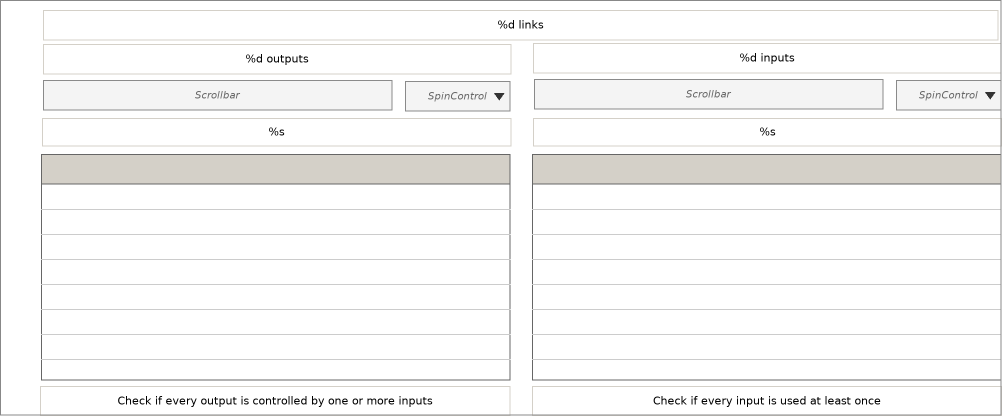
VISUALIZATION LinkInfo  // 1002x416
    Table (41,154 469x226), data array: MAIN.fbHome.stHmi.aLinkedInputs
        p3854506369: MAIN.fbHome.stHmi.aLinkedInputs[INDEX]
        p2232123230: Linked inputs
    Textfield (42,118 469x28), "%s", text variable: MAIN.fbHome.stHmi.sOutput
    SpinControl (405,81 105x30), variable: MAIN.fbHome.stHmi.nOutputIndex
        p651134158: MAIN.fbHome.fbDOGroupAll.nSize-1
    Scrollbar (43,80 349x30)
        p2245068023: MAIN.fbHome.fbDOGroupAll.nSize-1
        p1057716461: MAIN.fbHome.stHmi.nOutputIndex
    Textfield (533,118 469x28), "%s", text variable: MAIN.fbHome.stHmi.sInput
    Scrollbar (534,79 349x30)
        p2245068023: MAIN.fbHome.fbDIGroupAll.nSize-1
        p1057716461: MAIN.fbHome.stHmi.nInputIndex
    SpinControl (896,80 105x30), variable: MAIN.fbHome.stHmi.nInputIndex
        p651134158: MAIN.fbHome.fbDIGroupAll.nSize-1
    Table (532,154 469x226), data array: MAIN.fbHome.stHmi.aLinkedOutputs
        p3854506369: MAIN.fbHome.stHmi.aLinkedOutputs[INDEX]
        p2232123230: Linked outputs
    Textfield (43,10 955x30), "%d links", text variable: MAIN.fbHome.fbLinkManager.nSize
    Textfield (40,386 470x30), "Check if every output is controlled by one or more inputs"
    Textfield (532,386 470x30), "Check if every input is used at least once"
    Textfield (533,43 468x30), "%d inputs", text variable: MAIN.fbHome.fbDIGroupAll.nSize
    Textfield (43,44 468x30), "%d outputs", text variable: MAIN.fbHome.fbDOGroupAll.nSize
END_VISUALIZATION

(* stored: Version 1.1.0.1, ProductVersion 3.1.4024.12
   Visu LinkInfo: Id {0b9e9fec-83e7-4c47-a797-e13c82e18934} *)
